FUNCTION_BLOCK FB_ProductionMonitor IMPLEMENTS ITF_ProductionData
VAR CONSTANT
    //Constant declarations
    PRODUCTION_DATA_ALARM_COUNT : UDINT := 16;
END_VAR
VAR PERSISTENT
    //ITF_ProductionData internal variables
    tShiftLength             : TIME  := T#10M;
    nShiftProductionTarget   : DINT  := 1000;
    fWarningMargin           : LREAL := 10;
    fProductionRate_Setpoint : LREAL := 30;
    nRateAveragingCount      : DINT  := 10;
END_VAR
VAR
    //ITF_ProductionData internal variables + Other Production related variables
    bShiftComplete                    : BOOL;
    bProductComplete                  : BOOL;
    nCurrentShiftProductionCount      : INT;
    nCurrentShiftTarget               : DINT;
    tCurrentShiftTime                 : TIME;
    tRemainingShiftTime               : TIME;
    nCurrentWarningProductionCount    : DINT;
    nCurrentAcceptableProductionCount : DINT;

    fProductionRate_Required : LREAL;
    fProductionRate_Actual   : LREAL;

    a_nLastProductTimestamps  : ARRAY[1..100] OF ULINT; //Array of ULINT values (1 unit = 1ns) for the relative time of each of the last 100 completed products
    fbShiftTimer              : TON;
    fbProductComplete_RT      : R_TRIG;
    bNewProductionRate        : BOOL;
    fLastTargetProductionRate : LREAL;

    bResetMaxProductionCount   : BOOL;
    bResetTotalProductionCount : BOOL;

    nMaxProductionCount   : DINT;
    nTotalProductionCount : DINT;

    stProductionDataHMI          : ST_ProductionData_HMI;
    fbFIFO                       : FB_FIFO_ULINT_Array;
    a_fbProductionDataAlarms     : ARRAY[1..PRODUCTION_DATA_ALARM_COUNT] OF FB_TcAlarm;
    fTemp                        : LREAL;
    bInitialized                 : BOOL;
    initialize                   : INT;
    fLastProductionRate_Setpoint : LREAL;
END_VAR

PROPERTY CurrentShiftAcceptableProduction : DINT
GET
END_GET
SET
END_SET
END_PROPERTY

PROPERTY CurrentShiftProductionCount : DINT
GET
CurrentShiftProductionCount := nCurrentShiftProductionCount;
END_GET
END_PROPERTY

PROPERTY CurrentShiftTarget : DINT
GET
CurrentShiftTarget := nCurrentShiftTarget;
END_GET
END_PROPERTY

PROPERTY CurrentShiftTime : TIME
GET
CurrentShiftTime := tCurrentShiftTime;
END_GET
END_PROPERTY

PROPERTY CurrentShiftWarningProduction : DINT
GET
END_GET
SET
END_SET
END_PROPERTY

METHOD HMICommunication : BOOL
VAR_INPUT
END_VAR
//Production Data================================================================================================================================================

//Process HMI requests
IF stProductionDataHMI.bIncomingHMIRequest AND NOT stProductionDataHMI.bHMICommandConfirmation
    THEN //If a request has been issued by the HMI, and a previous request has not just E_SequenceState.Finished being processed
    IF stProductionDataHMI.bShiftProductionTargetHMISetRequest THEN
        nShiftProductionTarget                      := stProductionDataHMI.nShiftProductionTargetHMISetValue;
        stProductionDataHMI.bHMICommandConfirmation := TRUE; //Confirm that the request has been processed
    END_IF

    IF stProductionDataHMI.bWarningMarginHMISetRequest THEN
        fWarningMargin                              := stProductionDataHMI.fWarningMarginHMISetValue;
        stProductionDataHMI.bHMICommandConfirmation := TRUE; //Confirm that the request has been processed
    END_IF

    IF stProductionDataHMI.bShiftLengthHMISetRequest THEN
        tShiftLength                                := stProductionDataHMI.tShiftLengthHMISetValue;
        stProductionDataHMI.bHMICommandConfirmation := TRUE; //Confirm that the request has been processed
    END_IF

    IF stProductionDataHMI.bProductionRateHMISetRequest THEN
        fProductionRate_Setpoint                    := stProductionDataHMI.fProductionRateHMISetValue;
        stProductionDataHMI.bHMICommandConfirmation := TRUE; //Confirm that the request has been processed
    END_IF
END_IF

//Update HMI Status Info
stProductionDataHMI.tShiftLength                      := tShiftLength;
stProductionDataHMI.nShiftProductionTarget            := nShiftProductionTarget;
stProductionDataHMI.nCurrentShiftProductionCount      := nCurrentShiftProductionCount;
stProductionDataHMI.nCurrentShiftTarget               := nCurrentShiftTarget;
stProductionDataHMI.nCurrentAcceptableProductionCount := nCurrentAcceptableProductionCount;
stProductionDataHMI.nCurrentWarningProductionCount    := nCurrentWarningProductionCount;
stProductionDataHMI.tCurrentShiftTime                 := tCurrentShiftTime;
stProductionDataHMI.tRemainingShiftTime               := tRemainingShiftTime;
stProductionDataHMI.fProductionRate_Setpoint          := F_LREAL_RoundToPlace(fProductionRate_Setpoint, 1);
stProductionDataHMI.fProductionRate_Actual            := F_LREAL_RoundToPlace(fProductionRate_Actual, 1);
stProductionDataHMI.fProductionRate_Required          := F_LREAL_RoundToPlace(fProductionRate_Required, 1);
END_METHOD

METHOD initialize : BOOL
VAR_INPUT
END_VAR
END_METHOD

METHOD Monitor : BOOL
VAR_INPUT
END_VAR
IF NOT bInitialized THEN
    initialize();
    bInitialized := TRUE;
END_IF

fbFIFO(a_FIFO := a_nLastProductTimestamps);

fbShiftTimer(IN := NOT bShiftComplete, PT := tShiftLength, Q => bShiftComplete, ET => tCurrentShiftTime);
tRemainingShiftTime := tShiftLength - tCurrentShiftTime;

IF TIME_TO_DINT(tRemainingShiftTime) > 0 THEN
    fProductionRate_Required :=
        DINT_TO_LREAL(nShiftProductionTarget - nCurrentShiftProductionCount) / (TIME_TO_LREAL(tRemainingShiftTime) / 1000 / 60);

    nCurrentAcceptableProductionCount := nCurrentShiftTarget;

    nCurrentWarningProductionCount :=
        nShiftProductionTarget
            - (LREAL_TO_DINT((fProductionRate_Actual * (1 + fWarningMargin / 100)) * (TIME_TO_LREAL(tRemainingShiftTime) / 1000 / 60)));

    IF nCurrentWarningProductionCount < 0 THEN
        nCurrentWarningProductionCount := 0;
    END_IF
END_IF

fbProductComplete_RT(CLK := bProductComplete);

IF fbProductComplete_RT.Q THEN
    nCurrentShiftProductionCount := nCurrentShiftProductionCount + 1;
    nTotalProductionCount        := nTotalProductionCount + 1;

    IF nCurrentShiftProductionCount > nMaxProductionCount THEN
        nMaxProductionCount := nCurrentShiftProductionCount;
    END_IF

    fbFIFO.AddEntry(nEntry := F_GetSystemTime());
END_IF

IF (fbFIFO.EntryCount > nRateAveragingCount) THEN
    fbFIFO.RemoveEntry();
END_IF

fTemp := (TIME_TO_LREAL(ULINT_TO_TIME(fbFIFO.LastInValue - fbFIFO.NextOutValue)) / 10000 / 1000 / 60);

IF fTemp > 0 AND fbFIFO.EntryCount > 1 THEN
    fProductionRate_Actual := F_LREAL_RoundToPlace(DINT_TO_LREAL(fbFIFO.EntryCount - 1) / fTemp, 2);
END_IF

IF TIME_TO_DINT(tShiftLength) > 0 THEN
    nCurrentShiftTarget := LREAL_TO_DINT((TIME_TO_LREAL(tCurrentShiftTime) / TIME_TO_LREAL(tShiftLength)) * DINT_TO_LREAL(nShiftProductionTarget));
END_IF

IF bShiftComplete THEN
    nCurrentShiftProductionCount := 0;
END_IF

IF bResetMaxProductionCount THEN
    nMaxProductionCount := nCurrentShiftProductionCount;
END_IF

IF bResetTotalProductionCount THEN
    nTotalProductionCount := 0;
END_IF

IF fProductionRate_Setpoint <> fLastTargetProductionRate THEN
    bNewProductionRate := TRUE;
ELSE
    bNewProductionRate := FALSE;
END_IF

fLastTargetProductionRate := fProductionRate_Setpoint;
END_METHOD

PROPERTY NewProductionRate : BOOL
GET
NewProductionRate := bNewProductionRate;
END_GET
END_PROPERTY

PROPERTY ProductComplete : BOOL
GET
ProductComplete := bProductComplete;
END_GET
SET
bProductComplete := ProductComplete;
END_SET
END_PROPERTY

PROPERTY ProductionRate_Actual : LREAL
GET
ProductionRate_Actual := fProductionRate_Actual;
END_GET
END_PROPERTY

PROPERTY ProductionRate_Required : LREAL
GET
ProductionRate_Required := fProductionRate_Required;
END_GET
SET
fProductionRate_Required := ProductionRate_Required;
END_SET
END_PROPERTY

PROPERTY ProductionRate_Setpoint : LREAL
GET
ProductionRate_Setpoint := fProductionRate_Setpoint;
END_GET
SET
fProductionRate_Setpoint := ProductionRate_Setpoint;
END_SET
END_PROPERTY

PROPERTY RateAveragingCount : DINT
GET
RateAveragingCount := nRateAveragingCount;
END_GET
SET
nRateAveragingCount := RateAveragingCount;
END_SET
END_PROPERTY

PROPERTY RemainingShiftTime : TIME
GET
END_GET
SET
END_SET
END_PROPERTY

PROPERTY ShiftComplete : BOOL
GET
ShiftComplete := bShiftComplete;
END_GET
END_PROPERTY

PROPERTY ShiftLength : TIME
GET
ShiftLength := tShiftLength;
END_GET
SET
tShiftLength := ShiftLength;
END_SET
END_PROPERTY

PROPERTY ShiftProductionTarget : DINT
GET
ShiftProductionTarget := nShiftProductionTarget;
END_GET
SET
nShiftProductionTarget := ShiftProductionTarget;
END_SET
END_PROPERTY

PROPERTY WarningMargin : LREAL
GET
WarningMargin := fWarningMargin;
END_GET
SET
fWarningMargin := WarningMargin;
END_SET
END_PROPERTY

END_FUNCTION_BLOCK

(* stored: Version 1.1.0.1, ProductVersion 3.1.4024.11
   POU FB_ProductionMonitor: Id {f8203f13-c671-4490-a2dc-5fb35f3230d2}, SpecialFunc None
   Folder 02_ITF_ProductionData: Id {af28e88d-58be-4cbf-8273-0d45dad302f8}
   Folder 01_Config: Id {8b4ae294-3055-480d-843a-05df49b8588e}
   Folder 02_Control: Id {0c3617e5-eeff-4661-be72-00cba2094584}
   Folder 03_Status: Id {b0ea0d58-bef1-45ce-b6ee-3e65d176ea26}
   Property CurrentShiftAcceptableProduction: Id {4a2d9f09-6355-4584-83d8-3df60e464aca}
   Get Get: Id {5127f6ae-8779-4d0a-883f-e3b05126315b}
   Set Set: Id {7e2bcba5-298e-4ecc-8263-5954c87663e7}
   Property CurrentShiftProductionCount: Id {2fde7753-5566-4e3d-a00c-fd69e227f6fc}
   Get Get: Id {929b3a38-56e3-4200-b27e-a66487be016c}
   Property CurrentShiftTarget: Id {4e772aab-50c3-425f-9d02-09b9df1a3761}
   Get Get: Id {92ff02ff-e0b9-450b-a741-fcae14652385}
   Property CurrentShiftTime: Id {2c6df43c-ac6a-4073-9c92-abc53bc36195}
   Get Get: Id {87ba0b6a-169d-49d0-8462-1636d1eefa03}
   Property CurrentShiftWarningProduction: Id {38b3ea72-1780-45e3-87e4-c1df7ce98e6b}
   Get Get: Id {74a13a54-f1c5-48af-a52d-958561038ee7}
   Set Set: Id {38c4b2eb-3848-42d5-8f6c-f36908f52378}
   Method HMICommunication: Id {79819f0f-3f34-4ffc-b778-70fa3ff512b1}
   Method initialize: Id {d2f32f7b-b879-4075-b8c8-f9521ac7d6cb}
   Method Monitor: Id {d6925783-f0c0-4d56-bd5f-b384a479d04f}
   Property NewProductionRate: Id {1c902ea6-4ab0-4956-baf5-69697e9b1692}
   Get Get: Id {fd22614a-f382-4118-b827-8fa49ee6d47b}
   Property ProductComplete: Id {d633f3ee-fc86-41bb-8542-703e85ac188a}
   Get Get: Id {ddfb2225-5c67-4528-86dd-d655923b4524}
   Set Set: Id {16f7d6cd-09bf-4bfb-bcd4-0a15c45580e9}
   Property ProductionRate_Actual: Id {fda4bd07-9b7f-4aa3-bc4b-21d9de284fc6}
   Get Get: Id {4aa2e610-c003-4d66-9739-8c15d83f3011}
   Property ProductionRate_Required: Id {cf9c27ec-c6e8-4bd2-9bdf-8d0a81297b2b}
   Get Get: Id {46f7acd1-7f57-40e0-9736-73e37293bbb4}
   Set Set: Id {f233e109-af34-4e3f-ae25-27eac1bd62e8}
   Property ProductionRate_Setpoint: Id {7dcf6047-7174-4fbf-9eb6-f8e814826907}
   Get Get: Id {1c4b77e2-d31b-41bc-b4cb-7f4179637522}
   Set Set: Id {0d271468-5385-4c72-8b13-6c65fe14a13a}
   Property RateAveragingCount: Id {d4647b91-369c-4122-9ae9-fecc94a5e20f}
   Get Get: Id {62064f0f-1880-4011-8342-6e3e81ae004e}
   Set Set: Id {328b41bf-3d2c-4322-be62-074feb97d012}
   Property RemainingShiftTime: Id {545c0285-9272-4a9a-ad37-8fcfe6c1098a}
   Get Get: Id {15551c08-f49c-459b-87a4-657563c52084}
   Set Set: Id {fe45ff6d-85d9-4520-bb0c-96cb2abd423c}
   Property ShiftComplete: Id {1ca7a8fb-4b3f-40c8-b34c-aafc97bab7de}
   Get Get: Id {ea8f3e5c-4017-4e5f-98a6-31123c0388d8}
   Property ShiftLength: Id {07a20480-c78b-451f-bd14-b96f87dd15c0}
   Get Get: Id {6531d2f2-d5d3-44c8-91cd-5ad945e27013}
   Set Set: Id {6de0f7a0-d113-4669-aa56-7aa023af46dc}
   Property ShiftProductionTarget: Id {4137c496-2f15-40fd-98f5-c35c0d7755c6}
   Get Get: Id {5dd269b1-4304-47d5-89a8-24524985aa0c}
   Set Set: Id {c2be9886-0159-4e19-8865-38537a287cdb}
   Property WarningMargin: Id {b733ec6c-cdba-4b8e-8ee3-dd56e2568e62}
   Get Get: Id {7a6115fa-2a27-47af-aa63-4ca7ab0fa7a8}
   Set Set: Id {ec66a605-94d0-4b3a-8693-6ed12689d41e} *)
